// TIA Portal project "Progetto_1_timer" (V16)

(* hardware
DEVICE "S7-1200 station_1"  S7-1200 Station
   slot 0: "Rack_0"  S7-1200 Rack  Rack  V1.0
   slot 1: "PLC_1"  CPU 1215C DC/DC/Rly  6ES7 215-1HG40-0XB0  V4.4
*)

// ===== PLC "PLC_1"  CPU 1215C DC/DC/Rly =====

VAR_GLOBAL   // PLC tag table "Default tag table"
   "Marcia" AT %I1.0 : Bool;
   "Emergenza" AT %I0.7 : Bool;
   "Start" AT %I1.1 : Bool;
   "Arresto" AT %I1.2 : Bool;
   "Macchina ON" AT %M0.0 : Bool;   // Macchina accesa
   "Avanti" AT %Q0.0 : Bool;
   "Indietro" AT %Q0.1 : Bool;
   "Spia macchina accesa" AT %Q0.6 : Bool;
   "fotocellula1" AT %I0.0 : Bool;
   "fotocellula 2" AT %I0.1 : Bool;
   "spia_avanti" AT %Q0.7 : Bool;
   "spia_indietro" AT %Q1.0 : Bool;
   "arrivato" AT %M0.1 : Bool;
   "ritornato" AT %M0.2 : Bool;
   "fine" AT %M0.3 : Bool;
   "reset" AT %M0.4 : Bool;
   "attesa" AT %M0.5 : Bool;
END_VAR

// folder: System blocks/Program resources

DATA_BLOCK "IEC_Counter_0_DB"   // DB1
{ S7_Optimized_Access := 'TRUE' }
AUTHOR : Simatic
FAMILY : IEC
NAME : CNTR
VERSION : 1.0
// stored: InstanceOfName IEC_COUNTER
"IEC_COUNTER"
BEGIN
END_DATA_BLOCK

DATA_BLOCK "IEC_Timer_0_DB"   // DB2
{ S7_Optimized_Access := 'TRUE' }
AUTHOR : Simatic
FAMILY : IEC
NAME : IEC_TMR
VERSION : 1.0
// stored: InstanceOfName IEC_TIMER
"IEC_TIMER"
BEGIN
END_DATA_BLOCK

// folder: (top level)

ORGANIZATION_BLOCK "Main"   // OB1, LAD, ProgramCycle
TITLE = "Main Program Sweep (Cycle)"
{ S7_Optimized_Access := 'TRUE' }
VERSION : 0.1
// macchina 1 avvio nastro trasportatore
   VAR_INPUT
      Initial_Call : Bool;   // Initial call of this OB
      Remanence : Bool;   // =True, if remanent data are available
   END_VAR
BEGIN

REGION Network 1: Macchina accesa
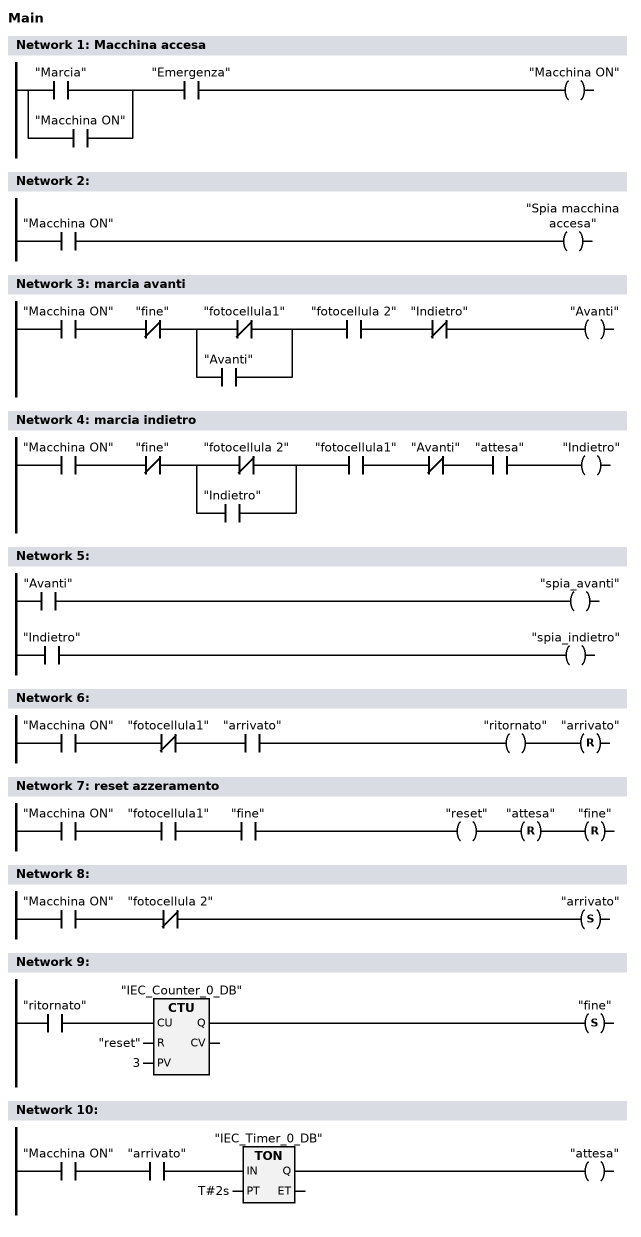
   RUNG wire#powerrail
      Contact( "Marcia" )
      wire#w1
      Contact( "Emergenza" )
      Coil( "Macchina ON" )
   END_RUNG
   RUNG wire#powerrail
      Contact( "Macchina ON" )
   END_RUNG wire#w1
   // the same network as SCL:
   "Macchina ON" := ("Marcia" OR "Macchina ON") AND "Emergenza";
END_REGION

REGION Network 2
   RUNG wire#powerrail
      Contact( "Macchina ON" )
      Coil( "Spia macchina accesa" )
   END_RUNG
   // the same network as SCL:
   "Spia macchina accesa" := "Macchina ON";
END_REGION

REGION Network 3: marcia avanti
   RUNG wire#powerrail
      Contact( "Macchina ON" )
      I_Contact( "fine" )
      wire#w1
      I_Contact( "fotocellula1" )
      wire#w2
      Contact( "fotocellula 2" )
      I_Contact( "Indietro" )
      Coil( "Avanti" )
   END_RUNG
   RUNG wire#w1
      Contact( "Avanti" )
   END_RUNG wire#w2
   // the same network as SCL:
   "Avanti" := "Macchina ON" AND NOT "fine" AND (NOT "fotocellula1" OR "Avanti") AND "fotocellula 2" AND NOT "Indietro";
END_REGION

REGION Network 4: marcia indietro
   RUNG wire#powerrail
      Contact( "Macchina ON" )
      I_Contact( "fine" )
      wire#w1
      I_Contact( "fotocellula 2" )
      wire#w2
      Contact( "fotocellula1" )
      I_Contact( "Avanti" )
      Contact( "attesa" )
      Coil( "Indietro" )
   END_RUNG
   RUNG wire#w1
      Contact( "Indietro" )
   END_RUNG wire#w2
   // the same network as SCL:
   "Indietro" := "Macchina ON" AND NOT "fine" AND (NOT "fotocellula 2" OR "Indietro") AND "fotocellula1" AND NOT "Avanti" AND "attesa";
END_REGION

REGION Network 5
   RUNG wire#powerrail
      Contact( "Avanti" )
      Coil( "spia_avanti" )
   END_RUNG
   RUNG wire#powerrail
      Contact( "Indietro" )
      Coil( "spia_indietro" )
   END_RUNG
   // the same network as SCL:
   "spia_avanti" := "Avanti";
   "spia_indietro" := "Indietro";
END_REGION

REGION Network 6
   RUNG wire#powerrail
      Contact( "Macchina ON" )
      I_Contact( "fotocellula1" )
      Contact( "arrivato" )
      Coil( "ritornato" )
      R_Coil( "arrivato" )
   END_RUNG
   // the same network as SCL:
   "ritornato" := "Macchina ON" AND NOT "fotocellula1" AND "arrivato";
   IF "ritornato" THEN "arrivato" := FALSE; END_IF;
END_REGION

REGION Network 7: reset azzeramento
   RUNG wire#powerrail
      Contact( "Macchina ON" )
      Contact( "fotocellula1" )
      Contact( "fine" )
      Coil( "reset" )
      R_Coil( "attesa" )
      R_Coil( "fine" )
   END_RUNG
   // the same network as SCL:
   "reset" := "Macchina ON" AND "fotocellula1" AND "fine";
   IF "reset" THEN
       "attesa" := FALSE;
       "fine" := FALSE;
   END_IF;
END_REGION

REGION Network 8
   RUNG wire#powerrail
      Contact( "Macchina ON" )
      I_Contact( "fotocellula 2" )
      S_Coil( "arrivato" )
   END_RUNG
   // the same network as SCL:
   IF "Macchina ON" AND NOT "fotocellula 2" THEN "arrivato" := TRUE; END_IF;
END_REGION

REGION Network 9
   "IEC_Counter_0_DB".CTU(CU := "ritornato", R := "reset", PV := 3);
   IF "IEC_Counter_0_DB".Q THEN "fine" := TRUE; END_IF;
END_REGION

REGION Network 10
   "IEC_Timer_0_DB".TON(IN := "Macchina ON" AND "arrivato", PT := T#2s);
   "attesa" := "IEC_Timer_0_DB".Q;
END_REGION
END_ORGANIZATION_BLOCK